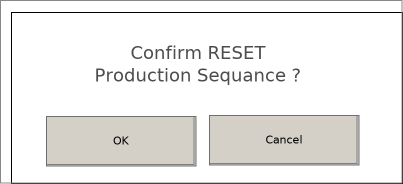
VISUALIZATION MSG_BOX_RESET  // 403x184
    RoundedRectangle (11,12 392x172)
    Button (46,116 150x50), "OK"
        OnMouseClick: execute {
            LOGFILE( sLogEvent	 := MSG.EVENT_BTN,
            		 sLogComp	 := MSG.COMP_HMI,
            		 sLogAction	 := MSG.ACTION_RESET,
            		 logFlag	 := TRUE);
            AUTO_MODE.Reset_seq_btn:= true;
        }
        OnMouseClick: CloseDialog Dialog=MSG_BOX_RESET, Result=OK, NumpadKeypadSet=True
    Button (209,115 150x50), "Cancel"
        OnMouseClick: CloseDialog Dialog=MSG_BOX_RESET, Result=Cancel, NumpadKeypadSet=True
    Label (80,20 236x88), "Confirm RESET Production Sequance ?"
END_VISUALIZATION

(* stored: Version 1.1.0.1, ProductVersion 3.1.4024.12
   Visu MSG_BOX_RESET: Id {80f6053b-b5f7-441e-81c8-5df6e4df20a7} *)
